(* IEC 61131-3 sources: Lasal/CPU_5344_V01/Class/closeClampsManual, 1 file *)

(* ---- closeClampsManual.st ---- *)
(*!
<Class
	Name               = "closeClampsManual"
	Revision           = "0.0"
	RealtimeTask       = "false"
	CyclicTask         = "false"
	BackgroundTask     = "false"
	Sigmatek           = "false"
	OSInterface        = "false"
	HighPriority       = "false"
	Automatic          = "false"
	UpdateMode         = "Prescan"
	SharedCommandTable = "true"
	Objectsize         = "(284,120)">
	<Channels>
		<Server Name="ClassSvr" Visualized="false" Initialize="false" WriteProtected="false" Retentive="false"/>
		<Client Name="ctrlCil" Required="true" Internal="false"/>
		<Client Name="oCmdhmi1" Required="true" Internal="false"/>
		<Client Name="oCmdhmi3" Required="true" Internal="false"/>
	</Channels>
</Class>
*)
closeClampsManual : CLASS
  //Servers:
	ClassSvr 	: SvrChCmd_DINT;
  //Clients:
	ctrlCil 	: CltChCmd_cmCil;
	oCmdhmi3 	: CltCh_eHMI_CmdPML;
	oCmdhmi1 	: CltCh_eHMI_CmdPML;
  //Variables:
  //Functions:

	FUNCTION VIRTUAL GLOBAL ClassSvr::Write
		VAR_INPUT
			input (EAX) 	: DINT;
		END_VAR
		VAR_OUTPUT
			result (EAX) 	: DINT;
		END_VAR;
  //Tables:
	FUNCTION @STD
		VAR_OUTPUT
			ret_code	: CONFSTATES;
		END_VAR;
	FUNCTION GLOBAL TAB @CT_;
END_CLASS;

#pragma usingLtd cmCil

FUNCTION VIRTUAL GLOBAL CloseClampsManual::ClassSvr::Write
	VAR_INPUT
		input (EAX) 	: DINT;
	END_VAR
	VAR_OUTPUT
		result (EAX) 	: DINT;
	END_VAR

	ClassSvr := input;

  IF ctrlCil.stsPos=cilIn THEN
    oCmdhmi3.Write(input:=cmd3);
  END_IF;

  IF ctrlCil.stsPos=cilOut | ctrlCil.stsPos = cilUnKnown THEN
    ocmdhmi1.write(input:=cmd1);
  END_IF;

	result := ClassSvr;

END_FUNCTION
